% RSLogix 500 project SENSOR CALIBRATION_BAK019.RSS, saved by version 8.30.00.16 %
PROJECT "UNTITLED"    % processor: Bul.1763 MicroLogix 1100 Series B %

PROGRAM FILES
  LAD 2 "MAIN"  4 rungs
  LAD 3 "OUTPUT"  3 rungs
  LAD 4 "CONTROLS"  5 rungs
  LAD 5 "CALIBR"  10 rungs

DATA FILES
  O0 OUTPUT  4 elements
  I1 INPUT  6 elements
  S2 STATUS  66 elements
  B3 BINARY  2 elements
  T4 TIMER  4 elements
  C5 COUNTER  1 elements
  R6 CONTROL  1 elements
  N7 INTEGER  15 elements
  F8 FLOAT  5 elements

LADDER 2 "MAIN"
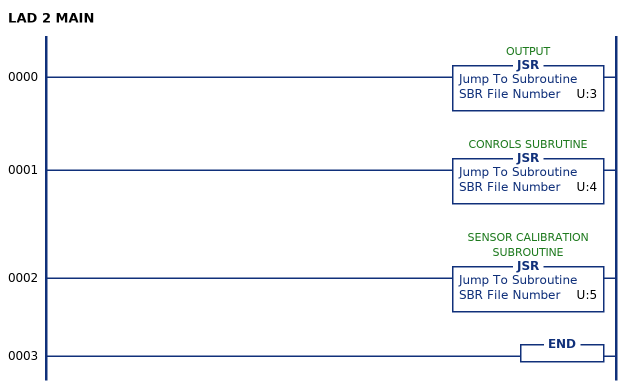
% Rung: 0 %
SOR JSR U:3 EOR
%   U:3  "OUTPUT" %
% Rung: 1 %
SOR JSR U:4 EOR
%   U:4  "CONROLS SUBRUTINE" %
% Rung: 2 %
SOR JSR U:5 EOR
%   U:5  "SENSOR CALIBRATION SUBROUTINE" %
% Rung: 3 %
SOR END EOR

LADDER 3 "OUTPUT"
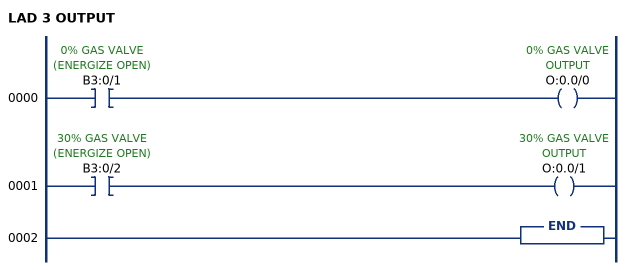
% Rung: 0 %
SOR XIC B3:0/1 OTE O:0.0/0 EOR
%   B3:0/1  "0% GAS VALVE (ENERGIZE OPEN)" %
%   O:0.0/0  "0% GAS VALVE OUTPUT" %
% Rung: 1 %
SOR XIC B3:0/2 OTE O:0.0/1 EOR
%   B3:0/2  "30% GAS VALVE (ENERGIZE OPEN)" %
%   O:0.0/1  "30% GAS VALVE OUTPUT" %
% Rung: 2 %
SOR END EOR

LADDER 4 "CONTROLS"
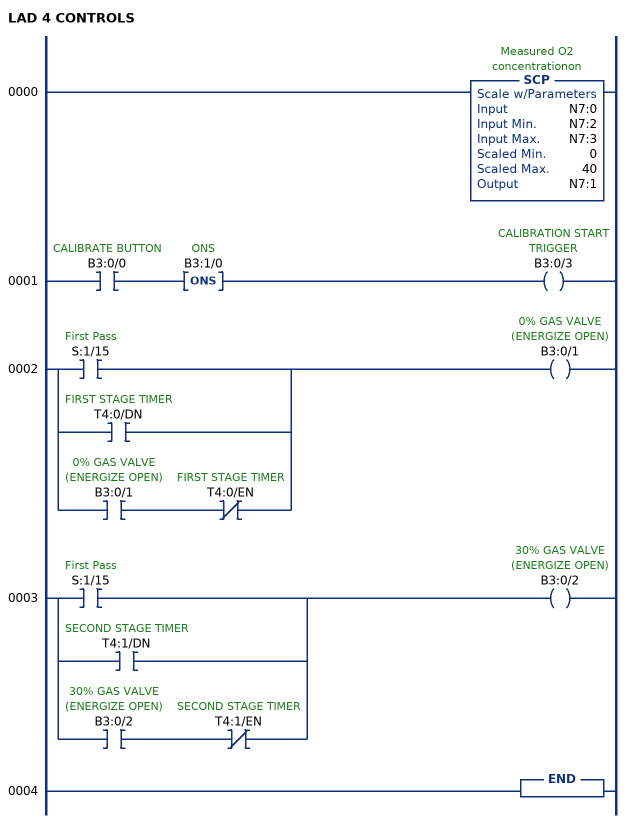
% Rung: 0 %
SOR SCP N7:0 N7:2 N7:3 0 40 N7:1 EOR
%   N7:0  "O2 sensor input signal" %
%   N7:2  "O2 input min (default = 0)" %
%   N7:3  "O2 input max (dafault = 16383)" %
%   N7:1  "Measured O2 concentrationon" %
% Rung: 1 %
SOR XIC B3:0/0 ONS B3:1/0 OTE B3:0/3 EOR
%   B3:0/0  "CALIBRATE BUTTON" %
%   B3:1/0  "ONS" %
%   B3:0/3  "CALIBRATION START TRIGGER" %
% Rung: 2 %
SOR BST XIC S:1/15 NXB XIC T4:0/DN NXB XIC B3:0/1 XIO T4:0/EN BND OTE B3:0/1 EOR
%   S:1/15  "First Pass" %
%   T4:0  "FIRST STAGE TIMER" %
%   B3:0/1  "0% GAS VALVE (ENERGIZE OPEN)" %
% Rung: 3 %
SOR BST XIC S:1/15 NXB XIC T4:1/DN NXB XIC B3:0/2 XIO T4:1/EN BND OTE B3:0/2 EOR
%   S:1/15  "First Pass" %
%   T4:1  "SECOND STAGE TIMER" %
%   B3:0/2  "30% GAS VALVE (ENERGIZE OPEN)" %
% Rung: 4 %
SOR END EOR

LADDER 5 "CALIBR"
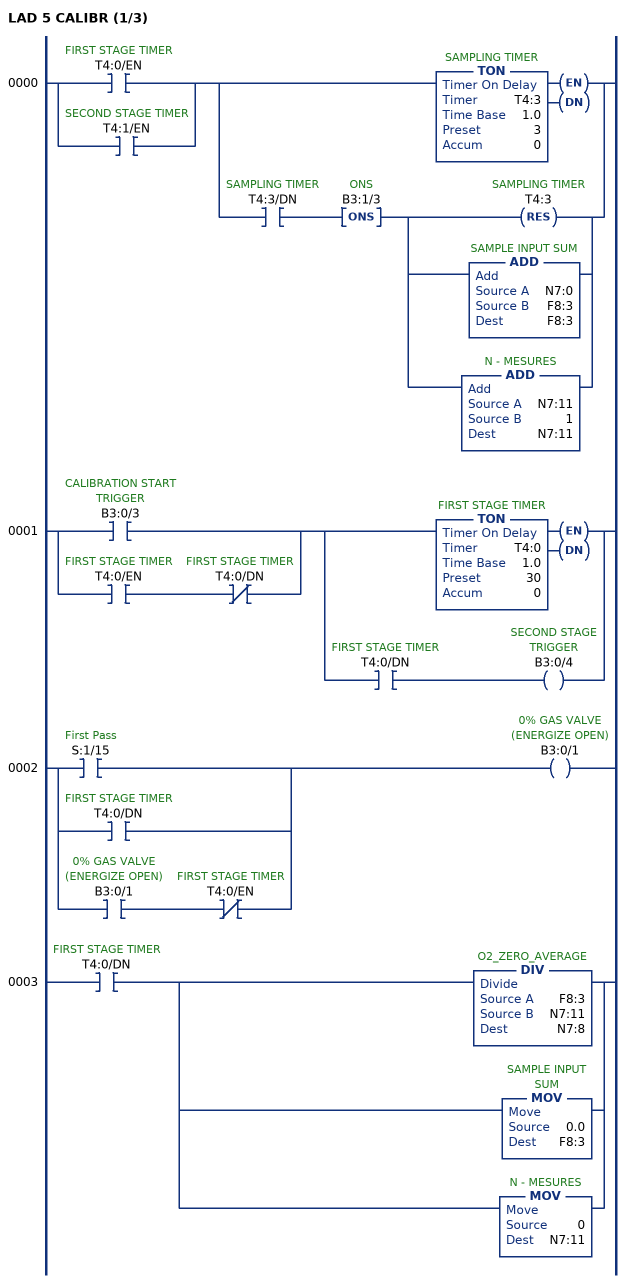
% Rung: 0 %
SOR BST XIC T4:0/EN NXB XIC T4:1/EN BND BST TON T4:3 1.0 3 0 NXB XIC T4:3/DN ONS B3:1/3 BST RES T4:3 NXB ADD N7:0 F8:3 F8:3 NXB ADD N7:11 1 N7:11 BND BND EOR
%   T4:0  "FIRST STAGE TIMER" %
%   T4:1  "SECOND STAGE TIMER" %
%   T4:3  "SAMPLING TIMER" %
%   B3:1/3  "ONS" %
%   N7:0  "O2 sensor input signal" %
%   F8:3  "SAMPLE INPUT SUM" %
%   N7:11  "N - MESURES" %
% Rung: 1 %
SOR BST XIC B3:0/3 NXB XIC T4:0/EN XIO T4:0/DN BND BST TON T4:0 1.0 30 0 NXB XIC T4:0/DN OTE B3:0/4 BND EOR
%   B3:0/3  "CALIBRATION START TRIGGER" %
%   T4:0  "FIRST STAGE TIMER" %
%   B3:0/4  "SECOND STAGE TRIGGER" %
% Rung: 2 %
SOR BST XIC S:1/15 NXB XIC T4:0/DN NXB XIC B3:0/1 XIO T4:0/EN BND OTE B3:0/1 EOR
%   S:1/15  "First Pass" %
%   T4:0  "FIRST STAGE TIMER" %
%   B3:0/1  "0% GAS VALVE (ENERGIZE OPEN)" %
% Rung: 3 %
SOR XIC T4:0/DN BST DIV F8:3 N7:11 N7:8 NXB MOV 0.0 F8:3 NXB MOV 0 N7:11 BND EOR
%   T4:0  "FIRST STAGE TIMER" %
%   F8:3  "SAMPLE INPUT SUM" %
%   N7:11  "N - MESURES" %
%   N7:8  "O2_ZERO_AVERAGE" %

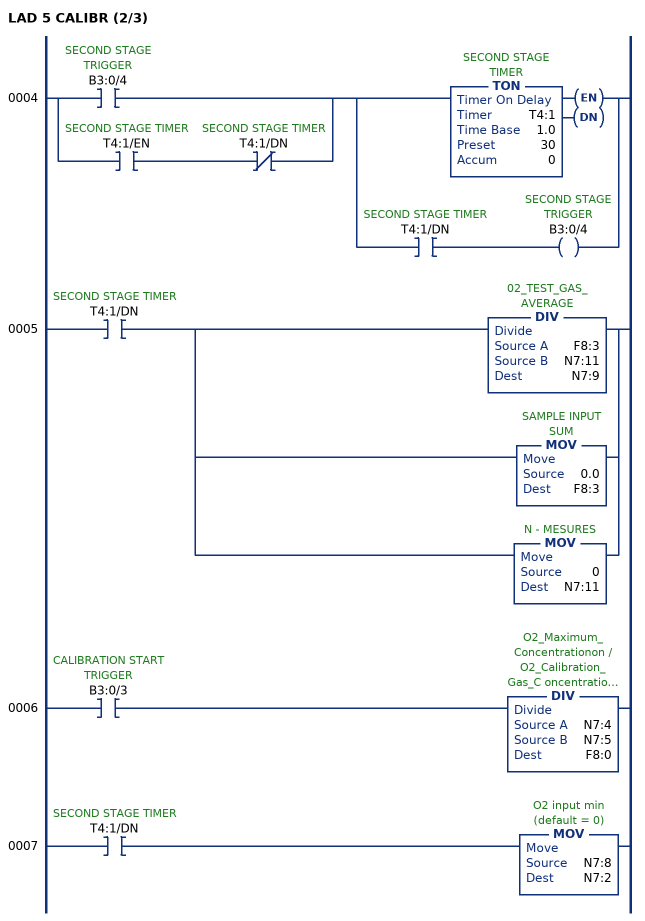
% Rung: 4 %
SOR BST XIC B3:0/4 NXB XIC T4:1/EN XIO T4:1/DN BND BST TON T4:1 1.0 30 0 NXB XIC T4:1/DN OTE B3:0/4 BND EOR
%   B3:0/4  "SECOND STAGE TRIGGER" %
%   T4:1  "SECOND STAGE TIMER" %
% Rung: 5 %
SOR XIC T4:1/DN BST DIV F8:3 N7:11 N7:9 NXB MOV 0.0 F8:3 NXB MOV 0 N7:11 BND EOR
%   T4:1  "SECOND STAGE TIMER" %
%   F8:3  "SAMPLE INPUT SUM" %
%   N7:11  "N - MESURES" %
%   N7:9  "02_TEST_GAS_AVERAGE" %
% Rung: 6 %
SOR XIC B3:0/3 DIV N7:4 N7:5 F8:0 EOR
%   B3:0/3  "CALIBRATION START TRIGGER" %
%   N7:4  "O2 MAX CONSENTRATION" %
%   N7:5  "O2 CONCENTRATION IN CALIBRATION GAS" %
%   F8:0  "O2_Maximum_ Concentrationon / O2_Calibration_Gas_C oncentratioon" %
% Rung: 7 %
SOR XIC T4:1/DN MOV N7:8 N7:2 EOR
%   T4:1  "SECOND STAGE TIMER" %
%   N7:8  "O2_ZERO_AVERAGE" %
%   N7:2  "O2 input min (default = 0)" %

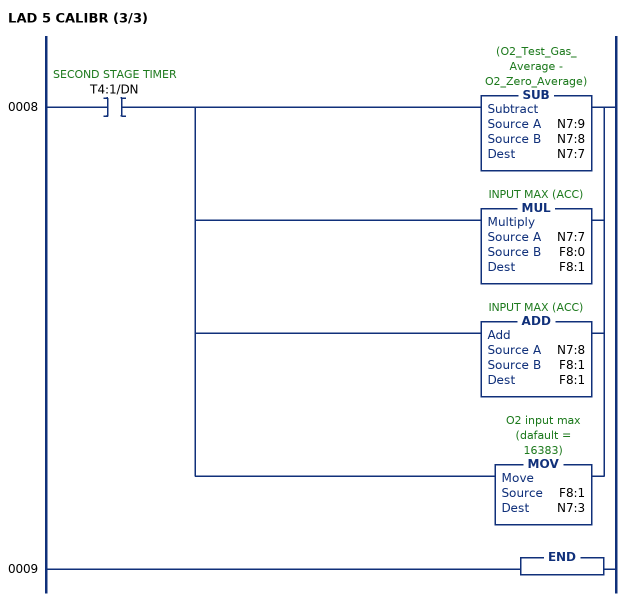
% Rung: 8 %
SOR XIC T4:1/DN BST SUB N7:9 N7:8 N7:7 NXB MUL N7:7 F8:0 F8:1 NXB ADD N7:8 F8:1 F8:1 NXB MOV F8:1 N7:3 BND EOR
%   T4:1  "SECOND STAGE TIMER" %
%   N7:9  "02_TEST_GAS_AVERAGE" %
%   N7:8  "O2_ZERO_AVERAGE" %
%   N7:7  "(O2_Test_Gas_Average - O2_Zero_Average)" %
%   F8:0  "O2_Maximum_ Concentrationon / O2_Calibration_Gas_C oncentratioon" %
%   F8:1  "INPUT MAX (ACC)" %
%   N7:3  "O2 input max (dafault = 16383)" %
% Rung: 9 %
SOR END EOR

OTHER DOCUMENTED ADDRESSES
  F8:2  "O2 sensor input signal / 1000"
  F8:4  "AVERAGE INPUT / 1000"
  N7:10  "SAMPLE INPUT SUM"

DATA TABLE (non-zero values as saved)
DATA B3
% B3:0 % 0X0006 0X0000
DATA T4
% .PRE .ACC %
% T4:0 % 30 0
% T4:1 % 30 0
% T4:3 % 3 0
DATA N7
% N7:0 % 100 0 100 14633 40 30 0 10900 100 11000
DATA F8
% F8:0 % 1.333333 14633.33 0 0 0
